FUNCTION_BLOCK FB_LsNcConveyer IMPLEMENTS  I_NcConveyer
VAR_INPUT
END_VAR
VAR_OUTPUT
END_VAR
VAR
	_Axis1	: AXIS_REF;
	_Axis2	: AXIS_REF;
END_VAR

{warning 'add property implementation'}
PROPERTY Axis1 : Tc2_MC2.AXIS_REF
GET
Axis1 := _Axis1;
END_GET
SET
_Axis1 := Axis1;
END_SET
END_PROPERTY

{warning 'add property implementation'}
PROPERTY Axis2 : Tc2_MC2.AXIS_REF
GET
Axis2 := _Axis2;
END_GET
SET
_Axis2 := Axis2;
END_SET
END_PROPERTY

{warning 'add method implementation '}
METHOD Execute : BOOL
ADSLOGSTR(ADSLOG_MSGTYPE_LOG,'Moving Long-Straight','');
END_METHOD

{warning 'add method implementation '}
METHOD Reset : BOOL
ADSLOGSTR(ADSLOG_MSGTYPE_LOG,'Reseting Long-Straight','');
END_METHOD

{warning 'add method implementation '}
METHOD Start : BOOL
ADSLOGSTR(ADSLOG_MSGTYPE_LOG,'Powering on Long-Straight','');
END_METHOD

{warning 'add method implementation '}
METHOD Stop : BOOL
ADSLOGSTR(ADSLOG_MSGTYPE_LOG,'Stopping Long-Straight','');
END_METHOD

END_FUNCTION_BLOCK

(* stored: Version 1.1.0.1, ProductVersion 3.1.4024.6
   POU FB_LsNcConveyer: Id {f8494908-811a-4147-8e99-dfe773f3f21a}, SpecialFunc None
   Property Axis1: Id {1a63d534-32e7-455b-822e-de5e691825df}
   Get Get: Id {ccd6ebd2-ca0d-4be4-9e5b-ecba35d3ddcd}
   Set Set: Id {7ea011ef-45ff-406a-b79c-d221a8ee607e}
   Property Axis2: Id {9c2f9899-0981-4938-a4b0-212eedfd04ef}
   Get Get: Id {6e434e26-17e1-4275-a641-5f52737578d1}
   Set Set: Id {2308371b-0827-4bd1-bb81-aa69dee69847}
   Method Execute: Id {23830e75-c0f1-421a-a62f-975e225b8db6}
   Method Reset: Id {817208e6-153b-4101-b4c3-5bcedf1ba8eb}
   Method Start: Id {8e0d8745-d3db-4ed1-b2dc-b482c1da8d15}
   Method Stop: Id {2337a735-a818-401f-8c32-bf763b66630b} *)
